{attribute 'GeneratedUsingTerminal: DL-EC1A-0000'}
{attribute addProperty BoxType "DL-EC1A-0000"}
{attribute addProperty Id "Tool_02_ScoreAT %I*DINT4"}
{attribute addProperty CRC "640120323"}
{attribute addProperty Size "4"}
TYPE ID04_Current_Value_26277603 EXTENDS InputBase_8311D824 :
STRUCT
	{attribute addProperty Name "Tool_02_Score"}
	Tool_02_Score AT %I* : DINT;
END_STRUCT
END_TYPE

(* stored: Version 1.1.0.1, ProductVersion 3.1.4024.12
   DUT ID04_Current_Value_26277603: Id {f03698ec-2c4d-0bef-0d33-a9cba222222f} *)
